Fanuc KAREL source: IO0216.KL

-- PROVISIONAL review KL for V770-1; original PC SHA256 223fec52eeb41adfea7c647d6f9c9a18b5ce391878b3f343e97b09857720947c
-- Incomplete behavior may be omitted. Consult companion uncertainty JSON. Do not deploy.
PROGRAM IO0216
%NOLOCKGROUP
-- UNRESOLVED_LOCAL_POOL 5 cells at code offset 13; source declarations unknown
-- DIRECT_LOCAL_WORD_ACCESS alone does not prove INTEGER, REAL, or BOOLEAN
BEGIN
  -- UNRESOLVED_PC offsets 0-18; opcodes 2B,2C,7B
  -- UNRESOLVED_PC offsets 23-30; opcodes 9D,23
  -- UNRESOLVED_PC offsets 35-49; opcodes 2E,22,9D,33,35
  -- UNRESOLVED_PC offsets 54-61; opcodes 9D,23
  -- UNRESOLVED_PC offsets 66-77; opcodes 2E,23
  -- UNRESOLVED_PC offsets 82-102; opcodes 22,9D,33,9D,33,36,4A
  -- UNRESOLVED_PC offsets 107-111; opcodes 7F
  -- UNRESOLVED_PC offsets 116-120; opcodes 27,AA
  -- UNRESOLVED_PC offsets 125-129; opcodes 7F
END IO0216
